PROGRAM P_SqlGeneratTestData
VAR
	
	fbSql : FB_EasySql;
	sSql : STRING(1000);
	sSqlInser : STRING(1000):='INSERT INTO myTable (myId,myCustomer,myValue) VALUES (1,$'Martin$',1.1),(2,$'Hans$',2.2),(3,$'Bjarne$',3.3),(4,$'Niels$',4.4),(5,$'Bo$',5.5),(6,$'Allan$',6.6),(7,$'Tom$',7.7),(8,$'Tom$',8.8),(9,$'Tom$',9.9),(10,$'Kurt$',10.1),(11,$'Kurt$',11.11)';	
		
	bDone : BOOL; //Command done
	bError : BOOL; //Command error
	sError : STRING(255);
	
	bStart : BOOL;
	iState : INT;
	
	
END_VAR

//Clean database and inserty test items.
CASE iState OF
	0:
		fbSql.pData := 0;
		fbSql.cbData := 0;
		fbSql.cbData := 0;
		fbSql.bExecute := FALSE;
		iState := 10;
		
	10:
		IF bStart THEN
			bStart := FALSE;
			iState := 100;
		END_IF
		
	100: // Truncate database
		sSql := 'DELETE FROM myTable'; //Normaly use TRUNCATE - but SqLite dont support TRUNCATE
		fbSql.pData := 0;
		fbSql.cbData := 0;
		fbSql.cbData := 0;
		fbSql.bExecute := TRUE;
		iState := 110;
		
	110:
		IF fbSql.bDone THEN
			fbSql.bExecute := FALSE;
			iState := 120;
		END_IF
		
	120:
		sSql := 'VACUUM'; //Normaly use TRUNCATE - but SqLite dont support TRUNCATE
		fbSql.bExecute := TRUE;
		iState := 130;
		
	130:
		IF NOT fbSql.bDone THEN
			fbSql.bExecute := FALSE;
			iState := 140;
		END_IF
		
	140:
		sSql := sSqlInser;
		fbSql.bExecute := TRUE;
		iState := 150;
		
	150:
		IF fbSql.bDone THEN
			iState := 0;
		END_IF
		


END_CASE



fbSql(
	bExecute:= , 
	wDBID:= 1, 
	pSql:= ADR(sSql), 
	cbSql:= SIZEOF(sSql), 
	pData:= , 
	cbData:= , 
	udiMaxOfRecord:= 0, 
	udiNoOfRecords=> , 
	bDone=> bDone, 
	bBusy=> , 
	bError=> bError, 
	sError=> sError);

END_PROGRAM

(* stored: Version 1.1.0.1, ProductVersion 3.1.4024.4
   POU P_SqlGeneratTestData: Id {346d790d-9874-4642-bc04-d94064a68e79}, SpecialFunc None *)
